PROGRAM MAIN
VAR
	fbController				: FB_Controller();
	fbLampOnOffAdapter			: FB_LampOnOffAdapter();
	fbLampSetDirectAdapter		: FB_LampSetDirectAdapter();
	fbLampUpDownAdapter			: FB_LampUpDownAdapter();
	fbLampSetDirectDALIAdapter	: FB_LampSetDirectDALIAdapter();	
	nSetLamp					: INT;
	bDimUp, bDimDown			: BOOL;
	bOff, bOn					: BOOL;
	nLightLevel					: BYTE;
END_VAR

CASE nSetLamp OF
	1:
		fbController.refActiveLamp REF= fbLampOnOffAdapter;
		nSetLamp := 0;
	2:
		fbController.refActiveLamp REF= fbLampSetDirectAdapter;
		nSetLamp := 0;
	3:
		fbController.refActiveLamp REF= fbLampUpDownAdapter;
		nSetLamp := 0;
	4:
		fbController.refActiveLamp REF= fbLampSetDirectDALIAdapter;
		nSetLamp := 0;
END_CASE

IF (__ISVALIDREF(fbController.refActiveLamp) AND_THEN fbController.refActiveLamp.bIsDALIDevice) THEN
	nLightLevel := TO_BYTE(fbController.fbActualValue.nValue * 100.0 / 254.0);
ELSE
	nLightLevel := fbController.fbActualValue.nValue;
END_IF

IF (bDimUp) THEN
	fbController.DimUp();
	bDimUp := FALSE;
END_IF

IF (bDimDown) THEN
	fbController.DimDown();
	bDimDown := FALSE;
END_IF

IF (bOff) THEN
	fbController.Off();
	bOff := FALSE;
END_IF

IF (bOn) THEN
	fbController.On();
	bOn := FALSE;
END_IF

END_PROGRAM

(* stored: Version 1.1.0.1, ProductVersion 3.1.4024.11
   POU MAIN: Id {ef33b4c1-c95d-4cf8-b9bf-7d346bd93484}, SpecialFunc None *)
